% RSLogix 500 project BARCODE.RSS, saved by version 8.30.00.16 %
PROJECT "UNTITLED"    % processor: Bul.1763 MicroLogix 1100 Series B %

PROGRAM FILES
  LAD 2 "MAIN"  15 rungs

DATA FILES
  O0 OUTPUT  4 elements
  I1 INPUT  6 elements
  S2 STATUS  66 elements
  B3 BINARY  1 elements
  T4 TIMER  1 elements
  C5 COUNTER  1 elements
  R6 CONTROL  1 elements
  N7 INTEGER  13 elements
  F8 FLOAT  1 elements
  ST9 STRING  10 elements

LADDER 2 "MAIN"
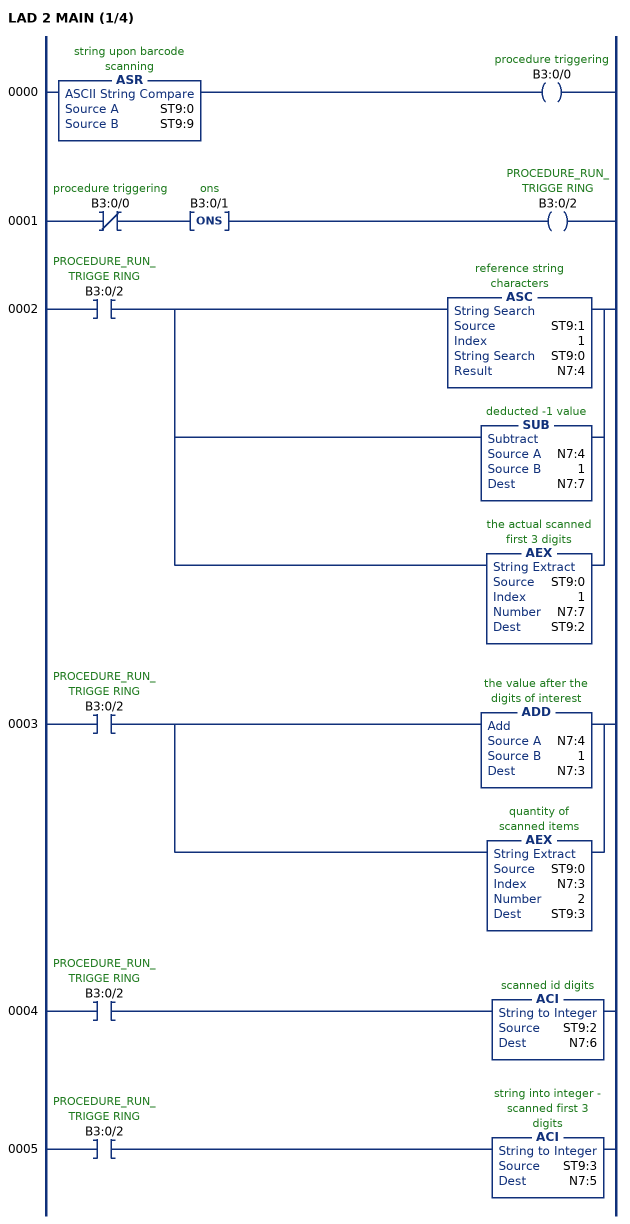
% Rung: 0 %
SOR ASR ST9:0 ST9:9 OTE B3:0/0 EOR
%   ST9:0  "string upon barcode scanning" %
%   ST9:9  "blank / empty / null / default value" %
%   B3:0/0  "procedure triggering" %
% Rung: 1 %
SOR XIO B3:0/0 ONS B3:0/1 OTE B3:0/2 EOR
%   B3:0/0  "procedure triggering" %
%   B3:0/1  "ons" %
%   B3:0/2  "PROCEDURE_RUN_TRIGGE RING" %
% Rung: 2 %
SOR XIC B3:0/2 BST ASC ST9:1 1 ST9:0 N7:4 NXB SUB N7:4 1 N7:7 NXB AEX ST9:0 1 N7:7 ST9:2 BND EOR
%   B3:0/2  "PROCEDURE_RUN_TRIGGE RING" %
%   ST9:1  "reference string characters" %
%   ST9:0  "string upon barcode scanning" %
%   N7:4  "location of dash" %
%   N7:7  "deducted -1 value" %
%   ST9:2  "the actual scanned first 3 digits" %
% Rung: 3 %
SOR XIC B3:0/2 BST ADD N7:4 1 N7:3 NXB AEX ST9:0 N7:3 2 ST9:3 BND EOR
%   B3:0/2  "PROCEDURE_RUN_TRIGGE RING" %
%   N7:4  "location of dash" %
%   N7:3  "the value after the digits of interest" %
%   ST9:0  "string upon barcode scanning" %
%   ST9:3  "quantity of scanned items" %
% Rung: 4 %
SOR XIC B3:0/2 ACI ST9:2 N7:6 EOR
%   B3:0/2  "PROCEDURE_RUN_TRIGGE RING" %
%   ST9:2  "the actual scanned first 3 digits" %
%   N7:6  "scanned id digits" %
% Rung: 5 %
SOR XIC B3:0/2 ACI ST9:3 N7:5 EOR
%   B3:0/2  "PROCEDURE_RUN_TRIGGE RING" %
%   ST9:3  "quantity of scanned items" %
%   N7:5  "string into integer - scanned first 3 digits" %

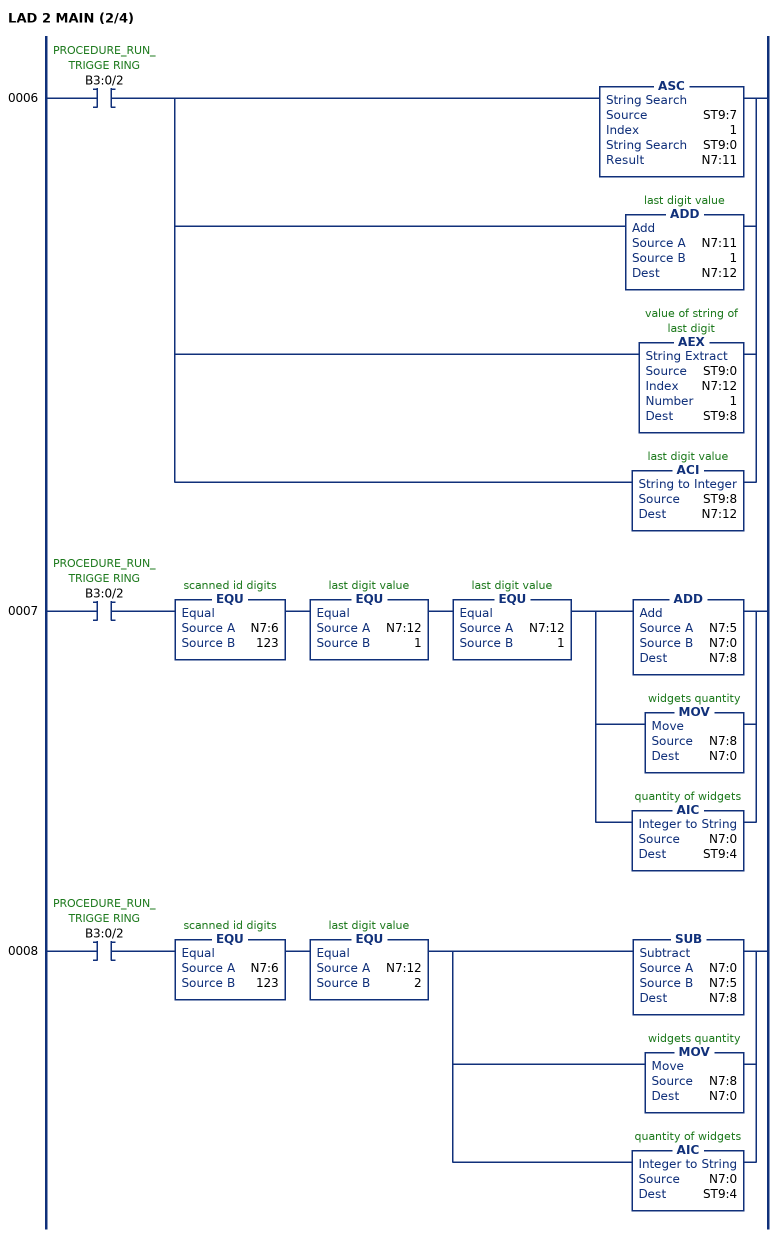
% Rung: 6 %
SOR XIC B3:0/2 BST ASC ST9:7 1 ST9:0 N7:11 NXB ADD N7:11 1 N7:12 NXB AEX ST9:0 N7:12 1 ST9:8 NXB ACI ST9:8 N7:12 BND EOR
%   B3:0/2  "PROCEDURE_RUN_TRIGGE RING" %
%   ST9:0  "string upon barcode scanning" %
%   N7:11  ": character for deduction or adding" %
%   N7:12  "last digit value" %
%   ST9:8  "value of string of last digit" %
% Rung: 7 %
SOR XIC B3:0/2 EQU N7:6 123 EQU N7:12 1 EQU N7:12 1 BST ADD N7:5 N7:0 N7:8 NXB MOV N7:8 N7:0 NXB AIC N7:0 ST9:4 BND EOR
%   B3:0/2  "PROCEDURE_RUN_TRIGGE RING" %
%   N7:6  "scanned id digits" %
%   N7:12  "last digit value" %
%   N7:5  "string into integer - scanned first 3 digits" %
%   N7:0  "widgets quantity" %
%   ST9:4  "quantity of widgets" %
% Rung: 8 %
SOR XIC B3:0/2 EQU N7:6 123 EQU N7:12 2 BST SUB N7:0 N7:5 N7:8 NXB MOV N7:8 N7:0 NXB AIC N7:0 ST9:4 BND EOR
%   B3:0/2  "PROCEDURE_RUN_TRIGGE RING" %
%   N7:6  "scanned id digits" %
%   N7:12  "last digit value" %
%   N7:0  "widgets quantity" %
%   N7:5  "string into integer - scanned first 3 digits" %
%   ST9:4  "quantity of widgets" %

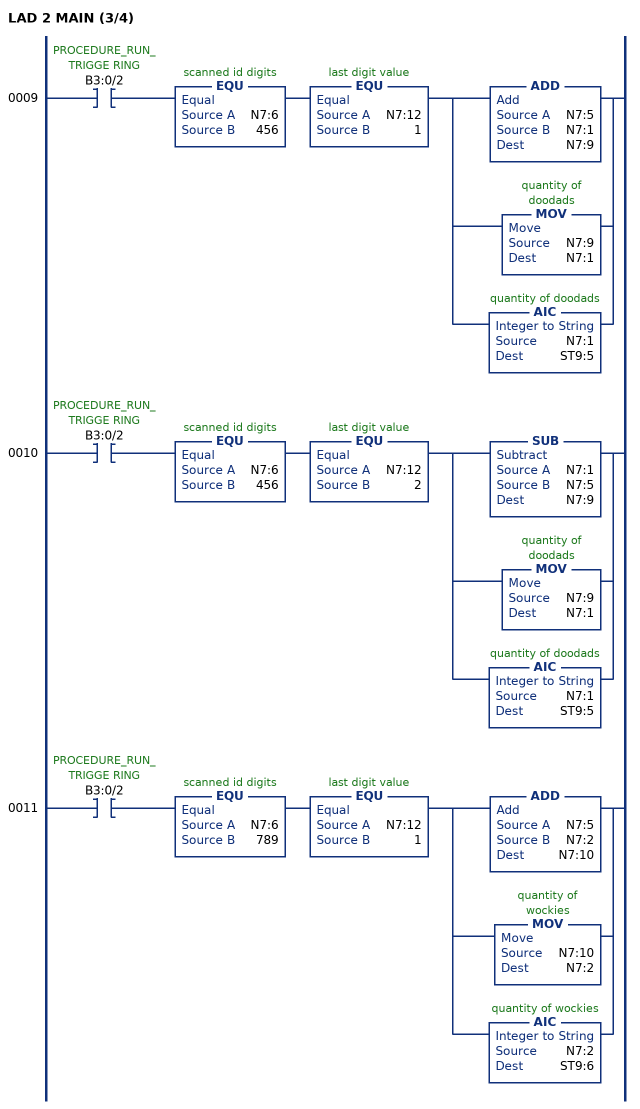
% Rung: 9 %
SOR XIC B3:0/2 EQU N7:6 456 EQU N7:12 1 BST ADD N7:5 N7:1 N7:9 NXB MOV N7:9 N7:1 NXB AIC N7:1 ST9:5 BND EOR
%   B3:0/2  "PROCEDURE_RUN_TRIGGE RING" %
%   N7:6  "scanned id digits" %
%   N7:12  "last digit value" %
%   N7:5  "string into integer - scanned first 3 digits" %
%   N7:1  "quantity of doodads" %
%   ST9:5  "quantity of doodads" %
% Rung: 10 %
SOR XIC B3:0/2 EQU N7:6 456 EQU N7:12 2 BST SUB N7:1 N7:5 N7:9 NXB MOV N7:9 N7:1 NXB AIC N7:1 ST9:5 BND EOR
%   B3:0/2  "PROCEDURE_RUN_TRIGGE RING" %
%   N7:6  "scanned id digits" %
%   N7:12  "last digit value" %
%   N7:1  "quantity of doodads" %
%   N7:5  "string into integer - scanned first 3 digits" %
%   ST9:5  "quantity of doodads" %
% Rung: 11 %
SOR XIC B3:0/2 EQU N7:6 789 EQU N7:12 1 BST ADD N7:5 N7:2 N7:10 NXB MOV N7:10 N7:2 NXB AIC N7:2 ST9:6 BND EOR
%   B3:0/2  "PROCEDURE_RUN_TRIGGE RING" %
%   N7:6  "scanned id digits" %
%   N7:12  "last digit value" %
%   N7:5  "string into integer - scanned first 3 digits" %
%   N7:2  "quantity of wockies" %
%   ST9:6  "quantity of wockies" %

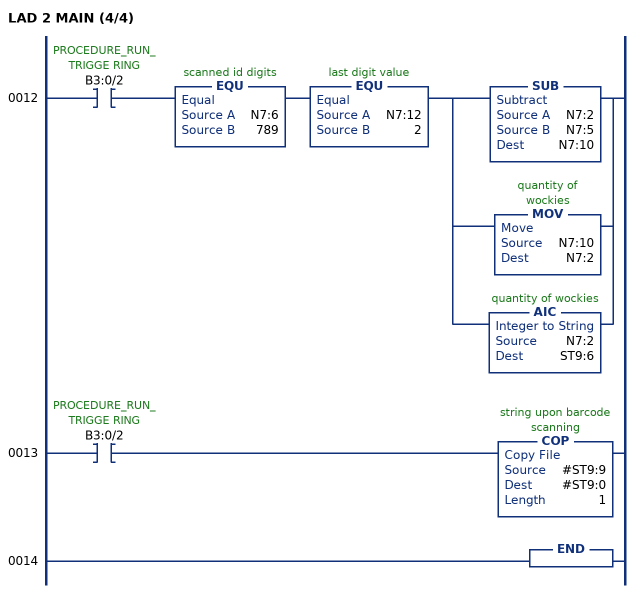
% Rung: 12 %
SOR XIC B3:0/2 EQU N7:6 789 EQU N7:12 2 BST SUB N7:2 N7:5 N7:10 NXB MOV N7:10 N7:2 NXB AIC N7:2 ST9:6 BND EOR
%   B3:0/2  "PROCEDURE_RUN_TRIGGE RING" %
%   N7:6  "scanned id digits" %
%   N7:12  "last digit value" %
%   N7:2  "quantity of wockies" %
%   N7:5  "string into integer - scanned first 3 digits" %
%   ST9:6  "quantity of wockies" %
% Rung: 13 %
SOR XIC B3:0/2 COP #ST9:9 #ST9:0 1 EOR
%   B3:0/2  "PROCEDURE_RUN_TRIGGE RING" %
%   ST9:9  "blank / empty / null / default value" %
%   ST9:0  "string upon barcode scanning" %
% Rung: 14 %
SOR END EOR

DATA TABLE (non-zero values as saved)
DATA B3
% B3:0 % 0X0001
DATA N7
% N7:0 % 0 0 0 5 4 1 456 3 0 0
% N7:10 % 0 7 2
DATA ST9
% ST9:1 % "-"
% ST9:2 % "456"
% ST9:3 % "01"
% ST9:4 % "0"
% ST9:5 % "0"
% ST9:6 % "0"
% ST9:7 % ":"
% ST9:8 % "2"
